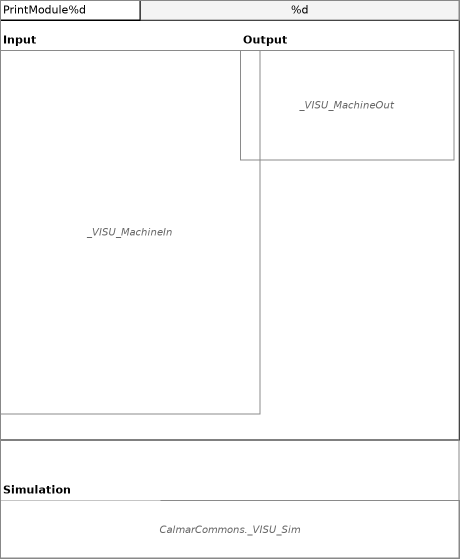
VISUALIZATION _VISU_MachineComm  // 460x559
VAR_IN_OUT
	mInst : FB_MachineComm;
END_VAR
    Rectangle (0,20 460x420)
    Frame (0,50 260x364)
        shows _VISU_MachineIn(ref := mInst.sModuleMachineState[mInst.nSelPm])
    Frame (240,50 214x110)
        shows _VISU_MachineOut(ref := mInst.sModuleMachineFeedback[mInst.nSelPm])
    Frame (0,500 460x59)
        shows CalmarCommons._VISU_Sim(mInst := mInst)
    Rectangle (240,30 160x20), "Output"
    Rectangle (0,30 160x20), "Input"
    Rectangle (0,480 160x20), "Simulation"
    Scrollbar (140,0 320x20), "%d", text variable: mInst.nSelPm
        p2245068023: iCPr_NB_PM
        p1057716461: mInst.nSelPm
    Rectangle (0,0 140x20), "PrintModule%d", text variable: PRG_PRINT.fbModuleMaster.nViewPmSel
END_VISUALIZATION

(* stored: Version 1.1.0.1, ProductVersion 3.1.4024.11
   Visu _VISU_MachineComm: Id {83823397-4c6b-4194-9438-b5cc85a44594} *)
